Staubli VAL3: pFrmCadToJoint.pgx

program pFrmCadToJoint(pointRx x_pTemp (dimensions=1), joint& x_jTemp[] (dimensions=1))
  local num l_ni
  local bool l_bTemp
begin
  ////  if strCmd=="RBINIT"
  //
  ////  endIf
  //    l_bTemp=pointToJoint(tTool,jConfig,x_pPtemp,x_jTemp)
  //  if l_bTemp==false
  //    //    io:socket="(RBERRO)"
  //    popUpMsg("wrong point position!!!")
  //  endIf
end
